(* Restituisce il numero del Pick-Point in cui è presente LA FALDA col codice desiderato, se restituisce -1, nessun Pick-Point ha il codice *)
FUNCTION TFPalletizerGetNumPickPointForLayerCode : UINT 
VAR_INPUT
	WorkPickPoint : POINTER TO ARRAY [1..MAXPICKPOINT] OF TFMachinePalletizer_WorkPickPointSlab;
	WorkPickPointState : POINTER TO ARRAY [1..MAXPICKPOINT] OF TFMachinePalletizer_WorkPickPoint_State;
	LayerCode : INT;
END_VAR
VAR
	pickpoint : UINT;
END_VAR

(* Restituisce il numero del Pick-Point in cui è presente LA FALDA col codice desiderato, se restituisce -1, nessun Pick-Point ha il codice *)
(* Per tutti i Pick-Point *)
FOR pickpoint:=1 TO MAXPICKPOINT DO
	(* Se il Pick Point è Abilitato *)
	IF WorkPickPoint^[pickpoint].Enable = 1 THEN
		(* Se il Pick Point è di tipo Magazzino Falde *)
		IF WorkPickPoint^[pickpoint].Tipologia = MAGAZZINO_FALDE THEN
			(* Se è presente almeno una falda *)
			IF WorkPickPointState^[WorkPickPoint^[pickpoint].ID].ProdPresence = PROD_PRESENTE THEN
				(* Se il codice coincide con quello richiesto *)
				IF WorkPickPointState^[WorkPickPoint^[pickpoint].ID].Code = LayerCode THEN
					(* La funzione restituisce il numero del Pick-Point *)
					TFPalletizerGetNumPickPointForLayerCode := (pickpoint);
					RETURN;
				END_IF	
			END_IF				
		END_IF
	END_IF
END_FOR
TFPalletizerGetNumPickPointForLayerCode := 0;

END_FUNCTION

(* stored: Version 1.1.0.1, ProductVersion 3.1.4024.11
   POU TFPalletizerGetNumPickPointForLayerCode: Id {94ea2132-b464-42da-80fa-00fe34948988}, SpecialFunc None *)
